(*Used as soft IO mapping to create a psuedo valve to communicate over two task on the same PLC.*) 
(*for FAST shutter control*)
FUNCTION_BLOCK FB_VFS_Interface
VAR_INPUT
	IG : ST_VG; // The Cold Cathode Data Structure
	{attribute 'pytmc' := '
    pv: FF_Reset
	'}
    i_xFFReset: BOOL;
END_VAR
VAR_IN_OUT

END_VAR
VAR

	(*outputs*)
	q_xPRESS_OK AT%Q*: BOOL;
	{attribute 'pytmc' := '
	pv: OPEN_SW; 
	field: ZNAM FALSE; 
	field: ONAM OPEN;
	io: io ;
	'}
	i_xOPN_SW AT%Q*:BOOL;
	{attribute 'pytmc' := '
	pv: CLS_SW; 
	field: ZNAM FALSE; 
	field: ONAM CLOSE;
	io: io ;
	'}
	q_xCLS_SW AT%Q*:BOOL; (*external open signal e.g epics*)
	{attribute 'pytmc' := '
	pv: FAULT_RESET; 
	field: ZNAM FALSE; 
	field: ONAM TRUE;
	io: io ;
	'}
	q_xVAC_FAULT_Reset AT%Q*: BOOL; (*Valve Vacuum OK, is set to False when there is Vacuum Fault*)
	{attribute 'pytmc' := '
	pv: VFS_OVRD_ON ;
	field: ZNAM Override OFF ;
	field: ONAM Override ON;
	io: io;
	'}
	i_xOverrideMode AT%Q*: BOOL; (*To be linked to global override bit. This Overrides Vacuum logic only, EPS, MPS and PMPS are still enforces*)
	{attribute 'pytmc' := '
    pv: VFS_FORCE_OPN;
	io: io;
	field: ZNAM FALSE;
	field: ONAM FORCE OPEN;
    '}
	i_xOverrideOpen AT%Q*: BOOL;
	
	(*inputs*)
	{attribute 'pytmc' := '
	pv: TRIG; 
	field: ZNAM TRIG_OFF; 
	field: ONAM TRIG_ON;
	io: io ;
	'}
	i_xTrigger AT %I* : BOOL;
	{attribute 'pytmc' := '
	pv: IS_OPEN; 
	field: ZNAM NOT OPEN; 
	field: ONAM OPEN;
	io: io ;
	'}
	i_xVFS_Open AT %I* : BOOL;
	{attribute 'pytmc' := '
	pv: IS_CLOSED; 
	field: ZNAM NOT CLOSED; 
	field: ONAM CLOSE;
	io: io ;
	'}
	i_xVFS_Closed AT %I* : BOOL;
	{attribute 'pytmc' := '
	pv: VAC_FAULT_OK; 
	field: ZNAM FAULT ; 
	field: ONAM FAULT OK;
	io: io ;
	'}
	i_xVAC_FAULT_OK AT%I*: BOOL; (*Valve Vacuum OK, is set to False when there is Vacuum Fault*)
	{attribute 'pytmc' := '
	pv: FFO_OK; 
	field: ZNAM FAULT ; 
	field: ONAM FAULT OK;
	io: io ;
	'}
	i_xMPS_OK AT%I*: BOOL;(*MPS Fault OK, is set when the Valve is Open and there is no trigger*)
END_VAR

(*soft IO Mapping*)

q_xPRESS_OK := IG.xPRESS_OK;

END_FUNCTION_BLOCK

(* stored: Version 1.1.0.1, ProductVersion 3.1.4022.18
   POU FB_VFS_Interface: Id {57bc9317-df03-4829-82d4-3e35e70264fe}, SpecialFunc None *)
